Fanuc KAREL source: kt00444.KL

-- PROVISIONAL review KL for V1013-1; original PC SHA256 f3847f90c5dfe53ced368f7c49dfa56eef6770df7e00d954604a5a39426fd70d
-- Incomplete behavior may be omitted. Consult companion uncertainty JSON. Do not deploy.
PROGRAM KT00444
%NOLOCKGROUP
VAR
  R1 : REAL
  OUT : BOOLEAN
-- UNRESOLVED_DECL H2 type=002017
BEGIN
  -- UNRESOLVED_PC offsets 5-16; opcodes 2E,23
  -- UNRESOLVED_PC offsets 21-35; opcodes 2E,22,9D,33,B4
  -- UNRESOLVED_PC offsets 40-63; opcodes 21,22,9D,33,B3,64,72,23
  -- UNRESOLVED_PC offsets 68-72; opcodes 7F
END KT00444
